(* PLC project SafeLOGIC-1, BrAutomation SafeDESIGNER  4.3.2.11 *)
(* stored: companyURL http://www.br-automation.com, creationDateTime Fri May 18 10:27:32 2018 *)

PROGRAM SafetyRun
  VAR  (* added by the conversion: wires and edge detectors of the diagram *)
    _OR_S82_OUT : SAFEBOOL;
  END_VAR

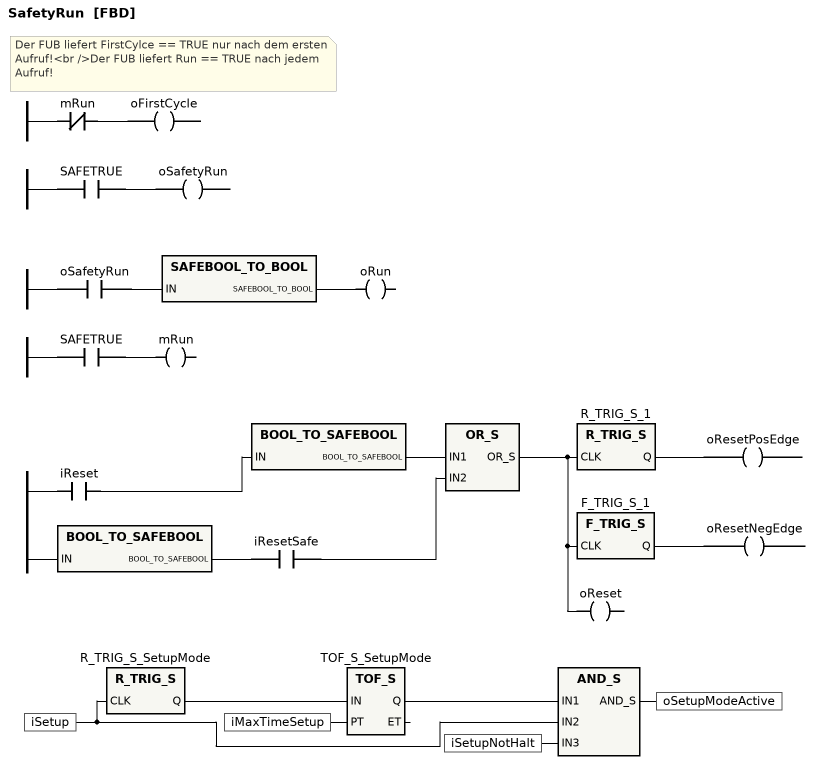
(* FBD diagram, written out as Structured Text *)
(* Der FUB liefert FirstCylce == TRUE nur nach dem ersten Aufruf!<br />Der FUB liefert Run == TRUE nach jedem Aufruf! *)
oFirstCycle := NOT mRun;
oSafetyRun := SAFETRUE;
oRun := SAFEBOOL_TO_BOOL(oSafetyRun);
mRun := SAFETRUE;
_OR_S82_OUT := OR_S(BOOL_TO_SAFEBOOL(iReset), BOOL_TO_SAFEBOOL(TRUE) AND iResetSafe);
R_TRIG_S_1(CLK := _OR_S82_OUT);
oResetPosEdge := R_TRIG_S_1.Q;
oReset := _OR_S82_OUT;
F_TRIG_S_1(CLK := _OR_S82_OUT);
oResetNegEdge := F_TRIG_S_1.Q;
R_TRIG_S_SetupMode(CLK := iSetup);
TOF_S_SetupMode(IN := R_TRIG_S_SetupMode.Q, PT := iMaxTimeSetup);
oSetupModeActive := AND_S(TOF_S_SetupMode.Q, iSetup, iSetupNotHalt);
END_PROGRAM
